# EPICS IOC start-up script: iocsh/ethercatmcPLCopenStateMachine.iocsh
ethercatmcCreateAsynParam $(MOTOR_PORT) PLCopenStateMachine Int32

dbLoadRecords("ethercatmcPLCopenStateMachine.template", "PREFIX=$(PREFIX), MOTOR_NAME=$(MOTOR_NAME), DESC=$(DESC), MOTOR_PORT=$(MOTOR_PORT), AXIS_NO=$(AXIS_NO), FB_NAME=PLCopenStateMachine")
